{attribute 'qualified_only'}
{attribute 'strict'}
TYPE EFeedbackMsgChamberBase :
(
	IsInMaintenanceMsg := 10,
	ArmNotExtendedMsg,
	EfemSlitDoorOpenPositionMsg,
	IsReadyToLoadUnloadMsg
);
END_TYPE

(* stored: Version 1.1.0.1, ProductVersion 3.1.4024.12
   DUT EFeedbackMsgChamberBase: Id {e51ba9f3-4d0b-4629-b529-456ae05d5837} *)
